TYPE ST_Machine:
STRUCT 
   rTemperature : REAL; 
   bRunning     : BOOL; 
END_STRUCT 
END_TYPE

(* stored: Version 1.1.0.1, ProductVersion 3.1.4024.16
   DUT ST_Machine: Id {e8ae8071-be8e-4abd-a09f-d932d3fa937e} *)
